// TIA Portal V20 export
DATA_BLOCK "InputData"   // DB1
TITLE = Dati in ingresso
{ S7_Optimized_Access := 'TRUE' }
AUTHOR : Nicola
// DB che raccogie di dati letti dai sensori in campo
// stored: MemoryReserve 100
   VAR
      Gt1IsClosed : Bool;   // Cancello 1 chiuso (False -> Aperto)
      Gt2IsClosed : Bool;   // Cancello 2 chiuso (False -> Aperto)
      Gt3IsClosed : Bool;   // Cancello 3 chiuso (False -> Aperto)
   END_VAR
BEGIN
END_DATA_BLOCK
